{attribute 'qualified_only'}
{attribute 'strict'}
{attribute 'to_string'}
TYPE
	E_Step :
	(
		Init := 0,
		Idel,
		Enable,
		MoveMoverstoSafePos,
		MoveMoversToStartPos,
		SetMasterPos,
		CamIn,
		MoveMasterToEndOfCam,
		MoveMasterToStartOfCam,
		AddAxisToCA,
		EnableCA,
		MoveSelectedMover,
		StoppingMaster,
		CamOut,
		HaltMovers,
		DisableCA,
		RemoveAxisFromCA,
		Disable,
		Error,
		Reset

	);
END_TYPE

(* stored: Version 1.1.0.1, ProductVersion 3.1.4024.12
   DUT E_Step: Id {9d1a9ace-f243-4597-824c-40153318b4c3} *)
